TYPE DUT_ObslugaAlarmow_Zdarzenie :
STRUCT
	sIdZdarzenia							: STRING [10];	//unikalny id zdarzenia x00x00x000
	byRodzaj								: BYTE;			//rodzaj zdarzenia błąd, ostrzerzenie, wiadomość, safety
	sOpis									: STRING;		//opis zdarzenia
	udiKod									: UDINT;		//kod błądu 
	bAktywny								: BOOL;			//czy aktywny
END_STRUCT
END_TYPE

(* stored: Version 1.1.0.1, ProductVersion 3.1.4024.11
   DUT DUT_ObslugaAlarmow_Zdarzenie: Id {c064e832-2d04-4b84-bc9b-a0b02cf89f41} *)
